{attribute addProperty BoxType "EK1100-0000-0018"}
{attribute addProperty Id "Beckhoff_EL4xxxEK1122Beckhoff_EL4xxxEK1122_E36AABB6162A_0001_EL4001_0000_0016EL4001_50B5189C9712.125A_0002_EL4001_0000_0017EL4001_50B5189C9712.125A_0003_EL4001_0000_0018EL4001_50B5189C9712.125A_0004_EL4001_0000_0019EL4001_50B5189C9712.125A_0005_EL4001_0000_0020EL4001_50B5189C9712.125A_0006_EL4002_0000_0016EL4002_19A75BD911314.125A_0007_EL4002_0000_0017EL4002_19A75BD911314.125A_0008_EL4002_0000_0018EL4002_BF483E0111314.125A_0009_EL4002_0000_0019EL4002_19A75BD911314.125A_0010_EL4002_0000_0020EL4002_19A75BD911314.125A_0011_EL4004_0000_0016EL4004_9786CACB14518.125A_0012_EL4004_0000_0017EL4004_9786CACB14518.125A_0013_EL4004_0000_0018EL4004_FEE36ED014518.125A_0014_EL4004_0000_0019EL4004_9786CACB14518.125A_0015_EL4004_0000_0020EL4004_9786CACB14518.125A_0016_EL4008_0000_0016EL4008_D5FA9EBB20926.125A_0017_EL4008_0000_0017EL4008_D5FA9EBB20926.125A_0018_EL4008_0000_0018EL4008_5F89906A20926.125A_0019_EL4008_0000_0019EL4008_D5FA9EBB20926.125A_0020_EL4008_0000_0020EL4008_D5FA9EBB20926.125A_0021_EL4011_0000_0016EL4011_50B5189C9712.125A_0022_EL4011_0000_0017EL4011_50B5189C9712.125A_0023_EL4011_0000_0018EL4011_50B5189C9712.125A_0024_EL4011_0000_0019EL4011_50B5189C9712.125A_0025_EL4011_0000_0020EL4011_50B5189C9712.125A_0026_EL4012_0000_0016EL4012_19A75BD911314.125A_0027_EL4012_0000_0017EL4012_19A75BD911314.125A_0028_EL4012_0000_0018EL4012_BF483E0111314.125A_0029_EL4012_0000_0019EL4012_19A75BD911314.125A_0030_EL4012_0000_0020EL4012_19A75BD911314.125A_0031_EL4014_0000_0016EL4014_9786CACB14518.125A_0032_EL4014_0000_0017EL4014_9786CACB14518.125A_0033_EL4014_0000_0018EL4014_FEE36ED014518.125A_0034_EL4014_0000_0019EL4014_9786CACB14518.125A_0035_EL4014_0000_0020EL4014_9786CACB14518.125A_0036_EL4018_0000_0016EL4018_D5FA9EBB20926.125A_0037_EL4018_0000_0017EL4018_D5FA9EBB20926.125A_0038_EL4018_0000_0018EL4018_5F89906A20926.125A_0039_EL4018_0000_0019EL4018_D5FA9EBB20926.125A_0040_EL4018_0000_0020EL4018_D5FA9EBB20926.125A_0041_EL4021_0000_0016EL4021_50B5189C9712.125A_0042_EL4021_0000_0017EL4021_50B5189C9712.125A_0043_EL4021_0000_0018EL4021_50B5189C9712.125A_0044_EL4021_0000_0019EL4021_50B5189C9712.125A_0045_EL4021_0000_0020EL4021_50B5189C9712.125A_0046_EL4021_0000_0021EL4021_50B5189C9712.125A_0047_EL4022_0000_0016EL4022_19A75BD911314.125A_0048_EL4022_0000_0017EL4022_19A75BD911314.125A_0049_EL4022_0000_0018EL4022_BF483E0111314.125A_0050_EL4022_0000_0019EL4022_19A75BD911314.125A_0051_EL4022_0000_0020EL4022_19A75BD911314.125A_0052_EL4022_0000_0021EL4022_19A75BD911314.125A_0053_EL4024_0000_0016EL4024_9786CACB14518.125A_0054_EL4024_0000_0017EL4024_9786CACB14518.125A_0055_EL4024_0000_0018EL4024_FEE36ED014518.125A_0056_EL4024_0000_0019EL4024_9786CACB14518.125A_0057_EL4024_0000_0020EL4024_9786CACB14518.125A_0058_EL4024_0000_0021EL4024_9786CACB14518.125A_0059_EL4028_0000_0016EL4028_D5FA9EBB20926.125A_0060_EL4028_0000_0017EL4028_D5FA9EBB20926.125A_0061_EL4028_0000_0018EL4028_5F89906A20926.125A_0062_EL4028_0000_0019EL4028_D5FA9EBB20926.125A_0063_EL4028_0000_0020EL4028_D5FA9EBB20926.125A_0064_EL4028_0000_0021EL4028_D5FA9EBB20926.125A_0065_EL4031_0000_0016EL4031_50B5189C9712.125A_0066_EL4031_0000_0017EL4031_50B5189C9712.125A_0067_EL4031_0000_0018EL4031_50B5189C9712.125A_0068_EL4031_0000_0019EL4031_50B5189C9712.125A_0069_EL4031_0000_0020EL4031_50B5189C9712.125A_0070_EL4032_0000_0016EL4032_19A75BD911314.125A_0071_EL4032_0000_0017EL4032_19A75BD911314.125A_0072_EL4032_0000_0018EL4032_BF483E0111314.125A_0073_EL4032_0000_0019EL4032_19A75BD911314.125A_0074_EL4032_0000_0020EL4032_19A75BD911314.125A_0075_EL4034_0000_0016EL4034_9786CACB14518.125A_0076_EL4034_0000_0017EL4034_9786CACB14518.125A_0077_EL4034_0000_0018EL4034_FEE36ED014518.125A_0078_EL4034_0000_0019EL4034_9786CACB14518.125A_0079_EL4034_0000_0020EL4034_9786CACB14518.125A_0080_EL4038_0000_0016EL4038_D5FA9EBB20926.125A_0081_EL4038_0000_0017EL4038_D5FA9EBB20926.125A_0082_EL4038_0000_0018EL4038_5F89906A20926.125A_0083_EL4038_0000_0019EL4038_D5FA9EBB20926.125A_0084_EL4038_0000_0020EL4038_D5FA9EBB20926.125A_0085_EL4102_0000_0000EL4102_6AE7330D11314.125A_0086_EL4102_0000_1016EL4102_6AE7330D11314.125A_0087_EL4102_0000_1017EL4102_6AE7330D11314.125A_0088_EL4102_0000_1018EL4102_6AE7330D11314.125A_0089_EL4102_0000_1019EL4102_6AE7330D11314.125A_0090_EL4102_0000_1020EL4102_6AE7330D11314.125A_0091_EL4104_0000_1016EL4104_FEE36ED014518.125A_0092_EL4104_0000_1017EL4104_FEE36ED014518.125A_0093_EL4104_0000_1018EL4104_FEE36ED014518.125A_0094_EL4104_0000_1019EL4104_FEE36ED014518.125A_0095_EL4104_0000_1020EL4104_FEE36ED014518.125A_0096_EL4112_0000_0000EL4112_6AE7330D11314.125A_0097_EL4112_0000_1016EL4112_6AE7330D11314.125A_0098_EL4112_0000_1017EL4112_6AE7330D11314.125A_0099_EL4112_0000_1018EL4112_6AE7330D11314.125A_0100_EL4112_0000_1019EL4112_6AE7330D11314.125A_0101_EL4112_0000_1020EL4112_6AE7330D11314.125A_0102_EL4112_0010_0000EL4112_6AE7330D11314.125A_0103_EL4112_0010_1016EL4112_6AE7330D11314.125A_0104_EL4112_0010_1017EL4112_6AE7330D11314.125A_0105_EL4112_0010_1018EL4112_6AE7330D11314.125A_0106_EL4112_0010_1019EL4112_6AE7330D11314.125A_0107_EL4112_0010_1020EL4112_6AE7330D11314.125A_0108_EL4114_0000_1016EL4114_FEE36ED014518.125A_0109_EL4114_0000_1017EL4114_FEE36ED014518.125A_0110_EL4114_0000_1018EL4114_FEE36ED014518.125A_0111_EL4114_0000_1019EL4114_FEE36ED014518.125A_0112_EL4114_0000_1020EL4114_FEE36ED014518.125A_0113_EL4122_0000_0000EL4122_6AE7330D11314.125A_0114_EL4122_0000_1016EL4122_6AE7330D11314.125A_0115_EL4122_0000_1017EL4122_6AE7330D11314.125A_0116_EL4122_0000_1018EL4122_6AE7330D11314.125A_0117_EL4122_0000_1019EL4122_6AE7330D11314.125A_0118_EL4122_0000_1020EL4122_6AE7330D11314.125A_0119_EL4124_0000_1016EL4124_FEE36ED014518.125A_0120_EL4124_0000_1017EL4124_FEE36ED014518.125A_0121_EL4124_0000_1018EL4124_FEE36ED014518.125A_0122_EL4124_0000_1019EL4124_FEE36ED014518.125A_0123_EL4124_0000_1020EL4124_FEE36ED014518.125A_0124_EL4132_0000_0000EL4132_6AE7330D11314.125A_0125_EL4132_0000_1016EL4132_6AE7330D11314.125A_0126_EL4132_0000_1017EL4132_6AE7330D11314.125A_0127_EL4132_0000_1018EL4132_6AE7330D11314.125A_0128_EL4132_0000_1019EL4132_6AE7330D11314.125A_0129_EL4132_0000_1020EL4132_6AE7330D11314.125A_0130_EL4134_0000_1016EL4134_FEE36ED014518.125A_0131_EL4134_0000_1017EL4134_FEE36ED014518.125A_0132_EL4134_0000_1018EL4134_FEE36ED014518.125A_0133_EL4134_0000_1019EL4134_FEE36ED014518.125A_0134_EL4134_0000_1020EL4134_FEE36ED014518.125A_0135_EL4134_0030_1020EL4134_FEE36ED014518.125"}
{attribute addProperty CRC "3023708240"}
{attribute addProperty SizeInBites "18295"}
{attribute addProperty SizeInBytes "2286.875"}
TYPE Beckhoff_EL4xxx_B43A2050 EXTENDS EK1100_179A0949 :
STRUCT
	{attribute addProperty Name "Beckhoff_EL4xxxEK1122"}
	Beckhoff_EL4xxxEK1122 : Beckhoff_EL4xxxEK1122_E36AABB6;
	{attribute addProperty Name "A_0001_EL4001_0000_0016"}
	A_0001_EL4001_0000_0016 : EL4001_50B5189C;
	{attribute addProperty Name "A_0002_EL4001_0000_0017"}
	A_0002_EL4001_0000_0017 : EL4001_50B5189C;
	{attribute addProperty Name "A_0003_EL4001_0000_0018"}
	A_0003_EL4001_0000_0018 : EL4001_50B5189C;
	{attribute addProperty Name "A_0004_EL4001_0000_0019"}
	A_0004_EL4001_0000_0019 : EL4001_50B5189C;
	{attribute addProperty Name "A_0005_EL4001_0000_0020"}
	A_0005_EL4001_0000_0020 : EL4001_50B5189C;
	{attribute addProperty Name "A_0006_EL4002_0000_0016"}
	A_0006_EL4002_0000_0016 : EL4002_19A75BD9;
	{attribute addProperty Name "A_0007_EL4002_0000_0017"}
	A_0007_EL4002_0000_0017 : EL4002_19A75BD9;
	{attribute addProperty Name "A_0008_EL4002_0000_0018"}
	A_0008_EL4002_0000_0018 : EL4002_BF483E01;
	{attribute addProperty Name "A_0009_EL4002_0000_0019"}
	A_0009_EL4002_0000_0019 : EL4002_19A75BD9;
	{attribute addProperty Name "A_0010_EL4002_0000_0020"}
	A_0010_EL4002_0000_0020 : EL4002_19A75BD9;
	{attribute addProperty Name "A_0011_EL4004_0000_0016"}
	A_0011_EL4004_0000_0016 : EL4004_9786CACB;
	{attribute addProperty Name "A_0012_EL4004_0000_0017"}
	A_0012_EL4004_0000_0017 : EL4004_9786CACB;
	{attribute addProperty Name "A_0013_EL4004_0000_0018"}
	A_0013_EL4004_0000_0018 : EL4004_FEE36ED0;
	{attribute addProperty Name "A_0014_EL4004_0000_0019"}
	A_0014_EL4004_0000_0019 : EL4004_9786CACB;
	{attribute addProperty Name "A_0015_EL4004_0000_0020"}
	A_0015_EL4004_0000_0020 : EL4004_9786CACB;
	{attribute addProperty Name "A_0016_EL4008_0000_0016"}
	A_0016_EL4008_0000_0016 : EL4008_D5FA9EBB;
	{attribute addProperty Name "A_0017_EL4008_0000_0017"}
	A_0017_EL4008_0000_0017 : EL4008_D5FA9EBB;
	{attribute addProperty Name "A_0018_EL4008_0000_0018"}
	A_0018_EL4008_0000_0018 : EL4008_5F89906A;
	{attribute addProperty Name "A_0019_EL4008_0000_0019"}
	A_0019_EL4008_0000_0019 : EL4008_D5FA9EBB;
	{attribute addProperty Name "A_0020_EL4008_0000_0020"}
	A_0020_EL4008_0000_0020 : EL4008_D5FA9EBB;
	{attribute addProperty Name "A_0021_EL4011_0000_0016"}
	A_0021_EL4011_0000_0016 : EL4011_50B5189C;
	{attribute addProperty Name "A_0022_EL4011_0000_0017"}
	A_0022_EL4011_0000_0017 : EL4011_50B5189C;
	{attribute addProperty Name "A_0023_EL4011_0000_0018"}
	A_0023_EL4011_0000_0018 : EL4011_50B5189C;
	{attribute addProperty Name "A_0024_EL4011_0000_0019"}
	A_0024_EL4011_0000_0019 : EL4011_50B5189C;
	{attribute addProperty Name "A_0025_EL4011_0000_0020"}
	A_0025_EL4011_0000_0020 : EL4011_50B5189C;
	{attribute addProperty Name "A_0026_EL4012_0000_0016"}
	A_0026_EL4012_0000_0016 : EL4012_19A75BD9;
	{attribute addProperty Name "A_0027_EL4012_0000_0017"}
	A_0027_EL4012_0000_0017 : EL4012_19A75BD9;
	{attribute addProperty Name "A_0028_EL4012_0000_0018"}
	A_0028_EL4012_0000_0018 : EL4012_BF483E01;
	{attribute addProperty Name "A_0029_EL4012_0000_0019"}
	A_0029_EL4012_0000_0019 : EL4012_19A75BD9;
	{attribute addProperty Name "A_0030_EL4012_0000_0020"}
	A_0030_EL4012_0000_0020 : EL4012_19A75BD9;
	{attribute addProperty Name "A_0031_EL4014_0000_0016"}
	A_0031_EL4014_0000_0016 : EL4014_9786CACB;
	{attribute addProperty Name "A_0032_EL4014_0000_0017"}
	A_0032_EL4014_0000_0017 : EL4014_9786CACB;
	{attribute addProperty Name "A_0033_EL4014_0000_0018"}
	A_0033_EL4014_0000_0018 : EL4014_FEE36ED0;
	{attribute addProperty Name "A_0034_EL4014_0000_0019"}
	A_0034_EL4014_0000_0019 : EL4014_9786CACB;
	{attribute addProperty Name "A_0035_EL4014_0000_0020"}
	A_0035_EL4014_0000_0020 : EL4014_9786CACB;
	{attribute addProperty Name "A_0036_EL4018_0000_0016"}
	A_0036_EL4018_0000_0016 : EL4018_D5FA9EBB;
	{attribute addProperty Name "A_0037_EL4018_0000_0017"}
	A_0037_EL4018_0000_0017 : EL4018_D5FA9EBB;
	{attribute addProperty Name "A_0038_EL4018_0000_0018"}
	A_0038_EL4018_0000_0018 : EL4018_5F89906A;
	{attribute addProperty Name "A_0039_EL4018_0000_0019"}
	A_0039_EL4018_0000_0019 : EL4018_D5FA9EBB;
	{attribute addProperty Name "A_0040_EL4018_0000_0020"}
	A_0040_EL4018_0000_0020 : EL4018_D5FA9EBB;
	{attribute addProperty Name "A_0041_EL4021_0000_0016"}
	A_0041_EL4021_0000_0016 : EL4021_50B5189C;
	{attribute addProperty Name "A_0042_EL4021_0000_0017"}
	A_0042_EL4021_0000_0017 : EL4021_50B5189C;
	{attribute addProperty Name "A_0043_EL4021_0000_0018"}
	A_0043_EL4021_0000_0018 : EL4021_50B5189C;
	{attribute addProperty Name "A_0044_EL4021_0000_0019"}
	A_0044_EL4021_0000_0019 : EL4021_50B5189C;
	{attribute addProperty Name "A_0045_EL4021_0000_0020"}
	A_0045_EL4021_0000_0020 : EL4021_50B5189C;
	{attribute addProperty Name "A_0046_EL4021_0000_0021"}
	A_0046_EL4021_0000_0021 : EL4021_50B5189C;
	{attribute addProperty Name "A_0047_EL4022_0000_0016"}
	A_0047_EL4022_0000_0016 : EL4022_19A75BD9;
	{attribute addProperty Name "A_0048_EL4022_0000_0017"}
	A_0048_EL4022_0000_0017 : EL4022_19A75BD9;
	{attribute addProperty Name "A_0049_EL4022_0000_0018"}
	A_0049_EL4022_0000_0018 : EL4022_BF483E01;
	{attribute addProperty Name "A_0050_EL4022_0000_0019"}
	A_0050_EL4022_0000_0019 : EL4022_19A75BD9;
	{attribute addProperty Name "A_0051_EL4022_0000_0020"}
	A_0051_EL4022_0000_0020 : EL4022_19A75BD9;
	{attribute addProperty Name "A_0052_EL4022_0000_0021"}
	A_0052_EL4022_0000_0021 : EL4022_19A75BD9;
	{attribute addProperty Name "A_0053_EL4024_0000_0016"}
	A_0053_EL4024_0000_0016 : EL4024_9786CACB;
	{attribute addProperty Name "A_0054_EL4024_0000_0017"}
	A_0054_EL4024_0000_0017 : EL4024_9786CACB;
	{attribute addProperty Name "A_0055_EL4024_0000_0018"}
	A_0055_EL4024_0000_0018 : EL4024_FEE36ED0;
	{attribute addProperty Name "A_0056_EL4024_0000_0019"}
	A_0056_EL4024_0000_0019 : EL4024_9786CACB;
	{attribute addProperty Name "A_0057_EL4024_0000_0020"}
	A_0057_EL4024_0000_0020 : EL4024_9786CACB;
	{attribute addProperty Name "A_0058_EL4024_0000_0021"}
	A_0058_EL4024_0000_0021 : EL4024_9786CACB;
	{attribute addProperty Name "A_0059_EL4028_0000_0016"}
	A_0059_EL4028_0000_0016 : EL4028_D5FA9EBB;
	{attribute addProperty Name "A_0060_EL4028_0000_0017"}
	A_0060_EL4028_0000_0017 : EL4028_D5FA9EBB;
	{attribute addProperty Name "A_0061_EL4028_0000_0018"}
	A_0061_EL4028_0000_0018 : EL4028_5F89906A;
	{attribute addProperty Name "A_0062_EL4028_0000_0019"}
	A_0062_EL4028_0000_0019 : EL4028_D5FA9EBB;
	{attribute addProperty Name "A_0063_EL4028_0000_0020"}
	A_0063_EL4028_0000_0020 : EL4028_D5FA9EBB;
	{attribute addProperty Name "A_0064_EL4028_0000_0021"}
	A_0064_EL4028_0000_0021 : EL4028_D5FA9EBB;
	{attribute addProperty Name "A_0065_EL4031_0000_0016"}
	A_0065_EL4031_0000_0016 : EL4031_50B5189C;
	{attribute addProperty Name "A_0066_EL4031_0000_0017"}
	A_0066_EL4031_0000_0017 : EL4031_50B5189C;
	{attribute addProperty Name "A_0067_EL4031_0000_0018"}
	A_0067_EL4031_0000_0018 : EL4031_50B5189C;
	{attribute addProperty Name "A_0068_EL4031_0000_0019"}
	A_0068_EL4031_0000_0019 : EL4031_50B5189C;
	{attribute addProperty Name "A_0069_EL4031_0000_0020"}
	A_0069_EL4031_0000_0020 : EL4031_50B5189C;
	{attribute addProperty Name "A_0070_EL4032_0000_0016"}
	A_0070_EL4032_0000_0016 : EL4032_19A75BD9;
	{attribute addProperty Name "A_0071_EL4032_0000_0017"}
	A_0071_EL4032_0000_0017 : EL4032_19A75BD9;
	{attribute addProperty Name "A_0072_EL4032_0000_0018"}
	A_0072_EL4032_0000_0018 : EL4032_BF483E01;
	{attribute addProperty Name "A_0073_EL4032_0000_0019"}
	A_0073_EL4032_0000_0019 : EL4032_19A75BD9;
	{attribute addProperty Name "A_0074_EL4032_0000_0020"}
	A_0074_EL4032_0000_0020 : EL4032_19A75BD9;
	{attribute addProperty Name "A_0075_EL4034_0000_0016"}
	A_0075_EL4034_0000_0016 : EL4034_9786CACB;
	{attribute addProperty Name "A_0076_EL4034_0000_0017"}
	A_0076_EL4034_0000_0017 : EL4034_9786CACB;
	{attribute addProperty Name "A_0077_EL4034_0000_0018"}
	A_0077_EL4034_0000_0018 : EL4034_FEE36ED0;
	{attribute addProperty Name "A_0078_EL4034_0000_0019"}
	A_0078_EL4034_0000_0019 : EL4034_9786CACB;
	{attribute addProperty Name "A_0079_EL4034_0000_0020"}
	A_0079_EL4034_0000_0020 : EL4034_9786CACB;
	{attribute addProperty Name "A_0080_EL4038_0000_0016"}
	A_0080_EL4038_0000_0016 : EL4038_D5FA9EBB;
	{attribute addProperty Name "A_0081_EL4038_0000_0017"}
	A_0081_EL4038_0000_0017 : EL4038_D5FA9EBB;
	{attribute addProperty Name "A_0082_EL4038_0000_0018"}
	A_0082_EL4038_0000_0018 : EL4038_5F89906A;
	{attribute addProperty Name "A_0083_EL4038_0000_0019"}
	A_0083_EL4038_0000_0019 : EL4038_D5FA9EBB;
	{attribute addProperty Name "A_0084_EL4038_0000_0020"}
	A_0084_EL4038_0000_0020 : EL4038_D5FA9EBB;
	{attribute addProperty Name "A_0085_EL4102_0000_0000"}
	A_0085_EL4102_0000_0000 : EL4102_6AE7330D;
	{attribute addProperty Name "A_0086_EL4102_0000_1016"}
	A_0086_EL4102_0000_1016 : EL4102_6AE7330D;
	{attribute addProperty Name "A_0087_EL4102_0000_1017"}
	A_0087_EL4102_0000_1017 : EL4102_6AE7330D;
	{attribute addProperty Name "A_0088_EL4102_0000_1018"}
	A_0088_EL4102_0000_1018 : EL4102_6AE7330D;
	{attribute addProperty Name "A_0089_EL4102_0000_1019"}
	A_0089_EL4102_0000_1019 : EL4102_6AE7330D;
	{attribute addProperty Name "A_0090_EL4102_0000_1020"}
	A_0090_EL4102_0000_1020 : EL4102_6AE7330D;
	{attribute addProperty Name "A_0091_EL4104_0000_1016"}
	A_0091_EL4104_0000_1016 : EL4104_FEE36ED0;
	{attribute addProperty Name "A_0092_EL4104_0000_1017"}
	A_0092_EL4104_0000_1017 : EL4104_FEE36ED0;
	{attribute addProperty Name "A_0093_EL4104_0000_1018"}
	A_0093_EL4104_0000_1018 : EL4104_FEE36ED0;
	{attribute addProperty Name "A_0094_EL4104_0000_1019"}
	A_0094_EL4104_0000_1019 : EL4104_FEE36ED0;
	{attribute addProperty Name "A_0095_EL4104_0000_1020"}
	A_0095_EL4104_0000_1020 : EL4104_FEE36ED0;
	{attribute addProperty Name "A_0096_EL4112_0000_0000"}
	A_0096_EL4112_0000_0000 : EL4112_6AE7330D;
	{attribute addProperty Name "A_0097_EL4112_0000_1016"}
	A_0097_EL4112_0000_1016 : EL4112_6AE7330D;
	{attribute addProperty Name "A_0098_EL4112_0000_1017"}
	A_0098_EL4112_0000_1017 : EL4112_6AE7330D;
	{attribute addProperty Name "A_0099_EL4112_0000_1018"}
	A_0099_EL4112_0000_1018 : EL4112_6AE7330D;
	{attribute addProperty Name "A_0100_EL4112_0000_1019"}
	A_0100_EL4112_0000_1019 : EL4112_6AE7330D;
	{attribute addProperty Name "A_0101_EL4112_0000_1020"}
	A_0101_EL4112_0000_1020 : EL4112_6AE7330D;
	{attribute addProperty Name "A_0102_EL4112_0010_0000"}
	A_0102_EL4112_0010_0000 : EL4112_6AE7330D;
	{attribute addProperty Name "A_0103_EL4112_0010_1016"}
	A_0103_EL4112_0010_1016 : EL4112_6AE7330D;
	{attribute addProperty Name "A_0104_EL4112_0010_1017"}
	A_0104_EL4112_0010_1017 : EL4112_6AE7330D;
	{attribute addProperty Name "A_0105_EL4112_0010_1018"}
	A_0105_EL4112_0010_1018 : EL4112_6AE7330D;
	{attribute addProperty Name "A_0106_EL4112_0010_1019"}
	A_0106_EL4112_0010_1019 : EL4112_6AE7330D;
	{attribute addProperty Name "A_0107_EL4112_0010_1020"}
	A_0107_EL4112_0010_1020 : EL4112_6AE7330D;
	{attribute addProperty Name "A_0108_EL4114_0000_1016"}
	A_0108_EL4114_0000_1016 : EL4114_FEE36ED0;
	{attribute addProperty Name "A_0109_EL4114_0000_1017"}
	A_0109_EL4114_0000_1017 : EL4114_FEE36ED0;
	{attribute addProperty Name "A_0110_EL4114_0000_1018"}
	A_0110_EL4114_0000_1018 : EL4114_FEE36ED0;
	{attribute addProperty Name "A_0111_EL4114_0000_1019"}
	A_0111_EL4114_0000_1019 : EL4114_FEE36ED0;
	{attribute addProperty Name "A_0112_EL4114_0000_1020"}
	A_0112_EL4114_0000_1020 : EL4114_FEE36ED0;
	{attribute addProperty Name "A_0113_EL4122_0000_0000"}
	A_0113_EL4122_0000_0000 : EL4122_6AE7330D;
	{attribute addProperty Name "A_0114_EL4122_0000_1016"}
	A_0114_EL4122_0000_1016 : EL4122_6AE7330D;
	{attribute addProperty Name "A_0115_EL4122_0000_1017"}
	A_0115_EL4122_0000_1017 : EL4122_6AE7330D;
	{attribute addProperty Name "A_0116_EL4122_0000_1018"}
	A_0116_EL4122_0000_1018 : EL4122_6AE7330D;
	{attribute addProperty Name "A_0117_EL4122_0000_1019"}
	A_0117_EL4122_0000_1019 : EL4122_6AE7330D;
	{attribute addProperty Name "A_0118_EL4122_0000_1020"}
	A_0118_EL4122_0000_1020 : EL4122_6AE7330D;
	{attribute addProperty Name "A_0119_EL4124_0000_1016"}
	A_0119_EL4124_0000_1016 : EL4124_FEE36ED0;
	{attribute addProperty Name "A_0120_EL4124_0000_1017"}
	A_0120_EL4124_0000_1017 : EL4124_FEE36ED0;
	{attribute addProperty Name "A_0121_EL4124_0000_1018"}
	A_0121_EL4124_0000_1018 : EL4124_FEE36ED0;
	{attribute addProperty Name "A_0122_EL4124_0000_1019"}
	A_0122_EL4124_0000_1019 : EL4124_FEE36ED0;
	{attribute addProperty Name "A_0123_EL4124_0000_1020"}
	A_0123_EL4124_0000_1020 : EL4124_FEE36ED0;
	{attribute addProperty Name "A_0124_EL4132_0000_0000"}
	A_0124_EL4132_0000_0000 : EL4132_6AE7330D;
	{attribute addProperty Name "A_0125_EL4132_0000_1016"}
	A_0125_EL4132_0000_1016 : EL4132_6AE7330D;
	{attribute addProperty Name "A_0126_EL4132_0000_1017"}
	A_0126_EL4132_0000_1017 : EL4132_6AE7330D;
	{attribute addProperty Name "A_0127_EL4132_0000_1018"}
	A_0127_EL4132_0000_1018 : EL4132_6AE7330D;
	{attribute addProperty Name "A_0128_EL4132_0000_1019"}
	A_0128_EL4132_0000_1019 : EL4132_6AE7330D;
	{attribute addProperty Name "A_0129_EL4132_0000_1020"}
	A_0129_EL4132_0000_1020 : EL4132_6AE7330D;
	{attribute addProperty Name "A_0130_EL4134_0000_1016"}
	A_0130_EL4134_0000_1016 : EL4134_FEE36ED0;
	{attribute addProperty Name "A_0131_EL4134_0000_1017"}
	A_0131_EL4134_0000_1017 : EL4134_FEE36ED0;
	{attribute addProperty Name "A_0132_EL4134_0000_1018"}
	A_0132_EL4134_0000_1018 : EL4134_FEE36ED0;
	{attribute addProperty Name "A_0133_EL4134_0000_1019"}
	A_0133_EL4134_0000_1019 : EL4134_FEE36ED0;
	{attribute addProperty Name "A_0134_EL4134_0000_1020"}
	A_0134_EL4134_0000_1020 : EL4134_FEE36ED0;
	{attribute addProperty Name "A_0135_EL4134_0030_1020"}
	A_0135_EL4134_0030_1020 : EL4134_FEE36ED0;
END_STRUCT
END_TYPE

(* stored: Version 1.2.0.0, ProductVersion 3.1.4024.9
   DUT Beckhoff_EL4xxx_B43A2050: Id {c976ffb8-0f35-4a95-9fb3-a74a2afac484} *)
